TYPE ST_CartMotorInput EXTENDS ST_MotorInputs :
STRUCT
	//
END_STRUCT
END_TYPE

(* stored: Version 1.1.0.1, ProductVersion 3.1.4024.12
   DUT ST_CartMotorInput: Id {590fb6f1-3bf5-4592-b6e1-ec7843cbfee6} *)
